FUNCTION_BLOCK AdapterTransition2 (* Template for an empty basic function block *)
  (* Standard: 61499-2; Description: Copyright (c) 2019 Jan Holzweber This program and the accompanying materials are made available under the terms of the Eclipse Public License 2.0 which is available at https://www.eclipse.org/legal/epl-2.0/ SPDX-License-Identifier: EPL-2.0 *)
  (* Version 1.0, 2019-06-21, Jan Holzweber *)
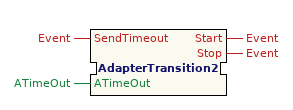
  EVENT_INPUT
    SendTimeout;
  END_EVENT
  EVENT_OUTPUT
    Start;
    Stop;
  END_EVENT
  SOCKETS
    ATimeOut : ATimeOut;
  END_SOCKETS
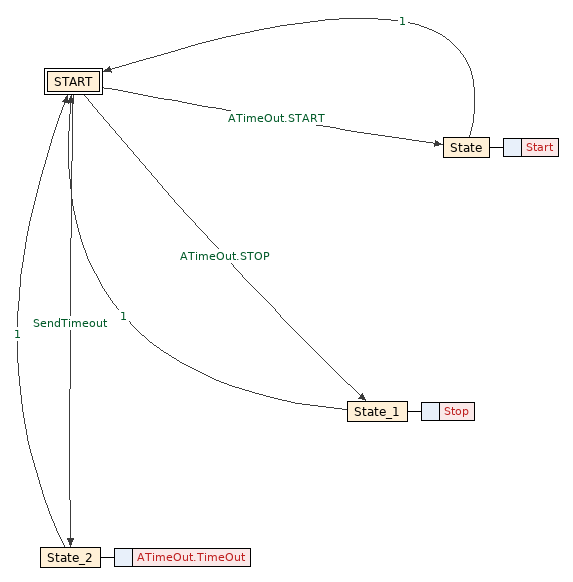
  EC_STATES
    START; (* Initial State *)
    State : -> Start;
    State_1 : -> Stop;
    State_2 : -> ATimeOut.TimeOut;
  END_STATES
  EC_TRANSITIONS
    START TO State := ATimeOut.START;
    State TO START := 1;
    START TO State_1 := ATimeOut.STOP;
    State_1 TO START := 1;
    START TO State_2 := SendTimeout;
    State_2 TO START := 1;
  END_TRANSITIONS
END_FUNCTION_BLOCK
